// TIA Portal V16 export
// export: Created 2021-07-12T14:47:20.353742Z, ExportSetting WithDefaults, DisplayName Totally Integrated Automation Portal, DisplayVersion V16, DisplayName TIA Portal Version Control Interface, DisplayVersion V16, DisplayName TIA Portal Openness, DisplayVersion V16, DisplayName STEP 7 Professional, DisplayVersion V16, DisplayName STEP 7 Safety, DisplayVersion V16, DisplayName WinCC Professional, DisplayVersion V16
TYPE "SimaHydTO_typeAxesArray"
TITLE = SimaHydTO_typeAxesArray
// Axis array of HMI axis selection
// stored: IsFailsafeCompliant false
   STRUCT
      axisData { ExternalAccessible := 'False'; ExternalVisible := 'False'; ExternalWritable := 'False'} : DB_ANY;   // DB number of hydraulic axis DB (HydAxisTO)
      basicControl { ExternalAccessible := 'False'; ExternalVisible := 'False'; ExternalWritable := 'False'; S7_SetPoint := 'True'} : "SimaHydTO_typeHMIConnectionBasicAxisControlCommand";   // HMI -> PLC: Axis commands of technology object via PLCopen functions
      directOutputControl { ExternalAccessible := 'False'; ExternalVisible := 'False'; ExternalWritable := 'False'; S7_SetPoint := 'True'} : "SimaHydTO_typeIHMIConnectionBasicAxisControlDirectOutput";
      VCharMeasurement { ExternalAccessible := 'False'; ExternalVisible := 'False'; ExternalWritable := 'False'; S7_SetPoint := 'True'} : "SimaHydTO_typeAxesArrayVCharMeasurement";
      advancedControl { ExternalAccessible := 'False'; ExternalVisible := 'False'; ExternalWritable := 'False'; S7_SetPoint := 'True'} : "SimaHydTO_typeHMIConnectionAdvancedAxisControlCommand";   // Advanced axis commands of technology object via PLCopen functions
      initialized { ExternalAccessible := 'False'; ExternalVisible := 'False'; ExternalWritable := 'False'} : Bool;   // Axis data initialized
   END_STRUCT;
END_TYPE
